// TIA Portal V19 export
DATA_BLOCK "LAF_InternalManual"   // DB43
VERSION : 19.0
// stored: MemoryReserve 100
   VAR
      hmi : Array[1..1] of "LAF_typeManHmiDisp";   // number of HMIs - modify the array size based on the required HMIs / nombre d'IHM - modifier la taille du tableau en fonction du nombre d'IHM requis / Anzahl der HMIs - modifizieren Sie die Array-Größe auf Basis der erforderlichen HMI / HMI 数量 - 根据所需的 HMI 修改数组大小
      manualOperationEnabled : Bool;   // feedback whether the manual operation lines are selected
   END_VAR
BEGIN
END_DATA_BLOCK
